PROGRAM PRG_PLAS_02_PackAggregationCtrl
VAR
	tonEnableCameraSystem					: TON;
	bEnablePackAggregationCameraSystem	: BOOL;
	bEnablePackTriggeringAfterDelay			: BOOL;

	tofPackAggregationCameraOFFDelay 		: TOF;
	rsInhibitCameraTrigger				: RS;
	rtrigNewArrived						: R_TRIG;
	bNewCodeIsProccesing				: BOOL;

	tonValidationTimout					: TON;
	bValidationTimeout					: BOOL;
	bValidationTimeoutReset				: BOOL;

	(*stPackAggregationCameraOptions		: ST_SCANNER_Options := (eScannerType := E_MV_420_FULL, nImageBuffer := 1, nExpectedResp := 1);*)
	fbPackAggregationCamera				: ARRAY [2..3] OF FB_SCANNER_CameraSelect;
	fbPackAggregationEvaluation			: ARRAY [2..3] OF FB_SCANNER_Evaluation;

	rtPackAggregationCameraDone		: ARRAY [2..3] OF R_TRIG;
	bPackAggregationCameraDone		: ARRAY [2..3] OF BOOL;

	fbAdd2PackToInfeedQ					: FB_T01_Add2PackToInfeedQ;
	(*bAddToPackQueueDone				: BOOL;*)

	fbDebugCNT							: FB_DEBUG_CounterArray;
	aCNTDebug							: ARRAY [1..10] OF UDINT;
	bResetCNT								: BOOL;

END_VAR
VAR // added by the converter: edge detectors and wires of the graphical bodies
    _w1 : BOOL;
    _w2 : UDINT;
END_VAR

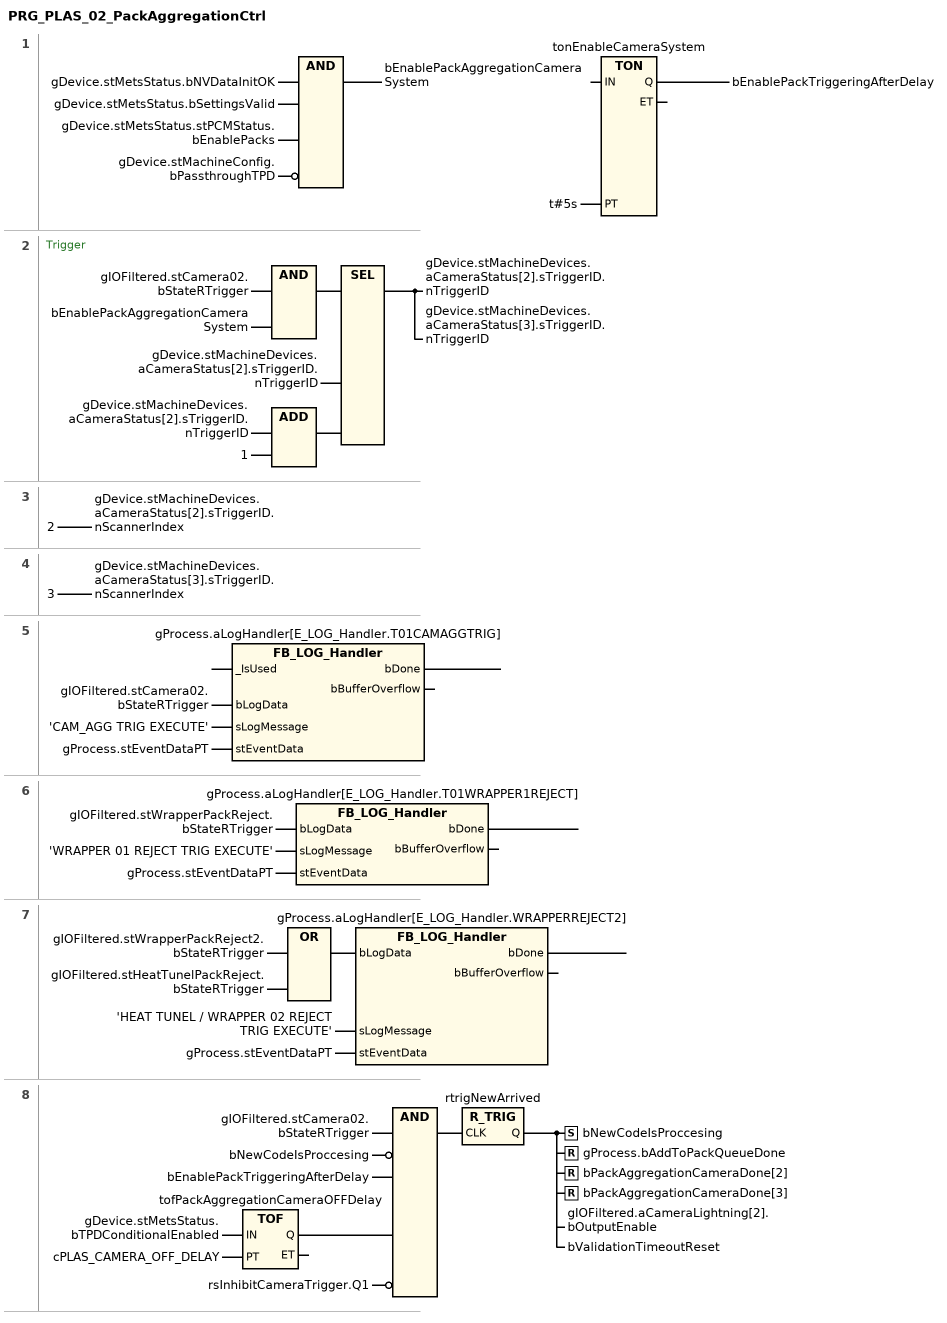
// NETWORK 1
_w1 := gDevice.stMetsStatus.bNVDataInitOK AND gDevice.stMetsStatus.bSettingsValid AND gDevice.stMetsStatus.stPCMStatus.bEnablePacks AND NOT gDevice.stMachineConfig.bPassthroughTPD;
bEnablePackAggregationCameraSystem := _w1;
tonEnableCameraSystem(IN := _w1, PT := t#5s); // TON
bEnablePackTriggeringAfterDelay := tonEnableCameraSystem.Q;

// NETWORK 2
// Trigger
_w2 := SEL(gIOFiltered.stCamera02.bStateRTrigger AND bEnablePackAggregationCameraSystem, gDevice.stMachineDevices.aCameraStatus[2].sTriggerID.nTriggerID, gDevice.stMachineDevices.aCameraStatus[2].sTriggerID.nTriggerID + 1);
gDevice.stMachineDevices.aCameraStatus[2].sTriggerID.nTriggerID := _w2;
gDevice.stMachineDevices.aCameraStatus[3].sTriggerID.nTriggerID := _w2;

// NETWORK 3
gDevice.stMachineDevices.aCameraStatus[2].sTriggerID.nScannerIndex := 2;

// NETWORK 4
gDevice.stMachineDevices.aCameraStatus[3].sTriggerID.nScannerIndex := 3;

// NETWORK 5
gProcess.aLogHandler[E_LOG_Handler.T01CAMAGGTRIG](
    bLogData := gIOFiltered.stCamera02.bStateRTrigger,
    sLogMessage := 'CAM_AGG TRIG EXECUTE',
    stEventData := gProcess.stEventDataPT); // FB_LOG_Handler

// NETWORK 6
gProcess.aLogHandler[E_LOG_Handler.T01WRAPPER1REJECT](
    bLogData := gIOFiltered.stWrapperPackReject.bStateRTrigger,
    sLogMessage := 'WRAPPER 01 REJECT TRIG EXECUTE',
    stEventData := gProcess.stEventDataPT); // FB_LOG_Handler

// NETWORK 7
gProcess.aLogHandler[E_LOG_Handler.WRAPPERREJECT2](
    bLogData := gIOFiltered.stWrapperPackReject2.bStateRTrigger OR gIOFiltered.stHeatTunelPackReject.bStateRTrigger,
    sLogMessage := 'HEAT TUNEL / WRAPPER 02 REJECT TRIG EXECUTE',
    stEventData := gProcess.stEventDataPT); // FB_LOG_Handler

// NETWORK 8
tofPackAggregationCameraOFFDelay(IN := gDevice.stMetsStatus.bTPDConditionalEnabled, PT := cPLAS_CAMERA_OFF_DELAY); // TOF
rtrigNewArrived(CLK := gIOFiltered.stCamera02.bStateRTrigger AND NOT bNewCodeIsProccesing AND bEnablePackTriggeringAfterDelay AND tofPackAggregationCameraOFFDelay.Q AND NOT rsInhibitCameraTrigger.Q1); // R_TRIG
bNewCodeIsProccesing S= rtrigNewArrived.Q;
gProcess.bAddToPackQueueDone R= rtrigNewArrived.Q;
bPackAggregationCameraDone[2] R= rtrigNewArrived.Q;
bPackAggregationCameraDone[3] R= rtrigNewArrived.Q;
gIOFiltered.aCameraLightning[2].bOutputEnable := rtrigNewArrived.Q;
bValidationTimeoutReset := rtrigNewArrived.Q;

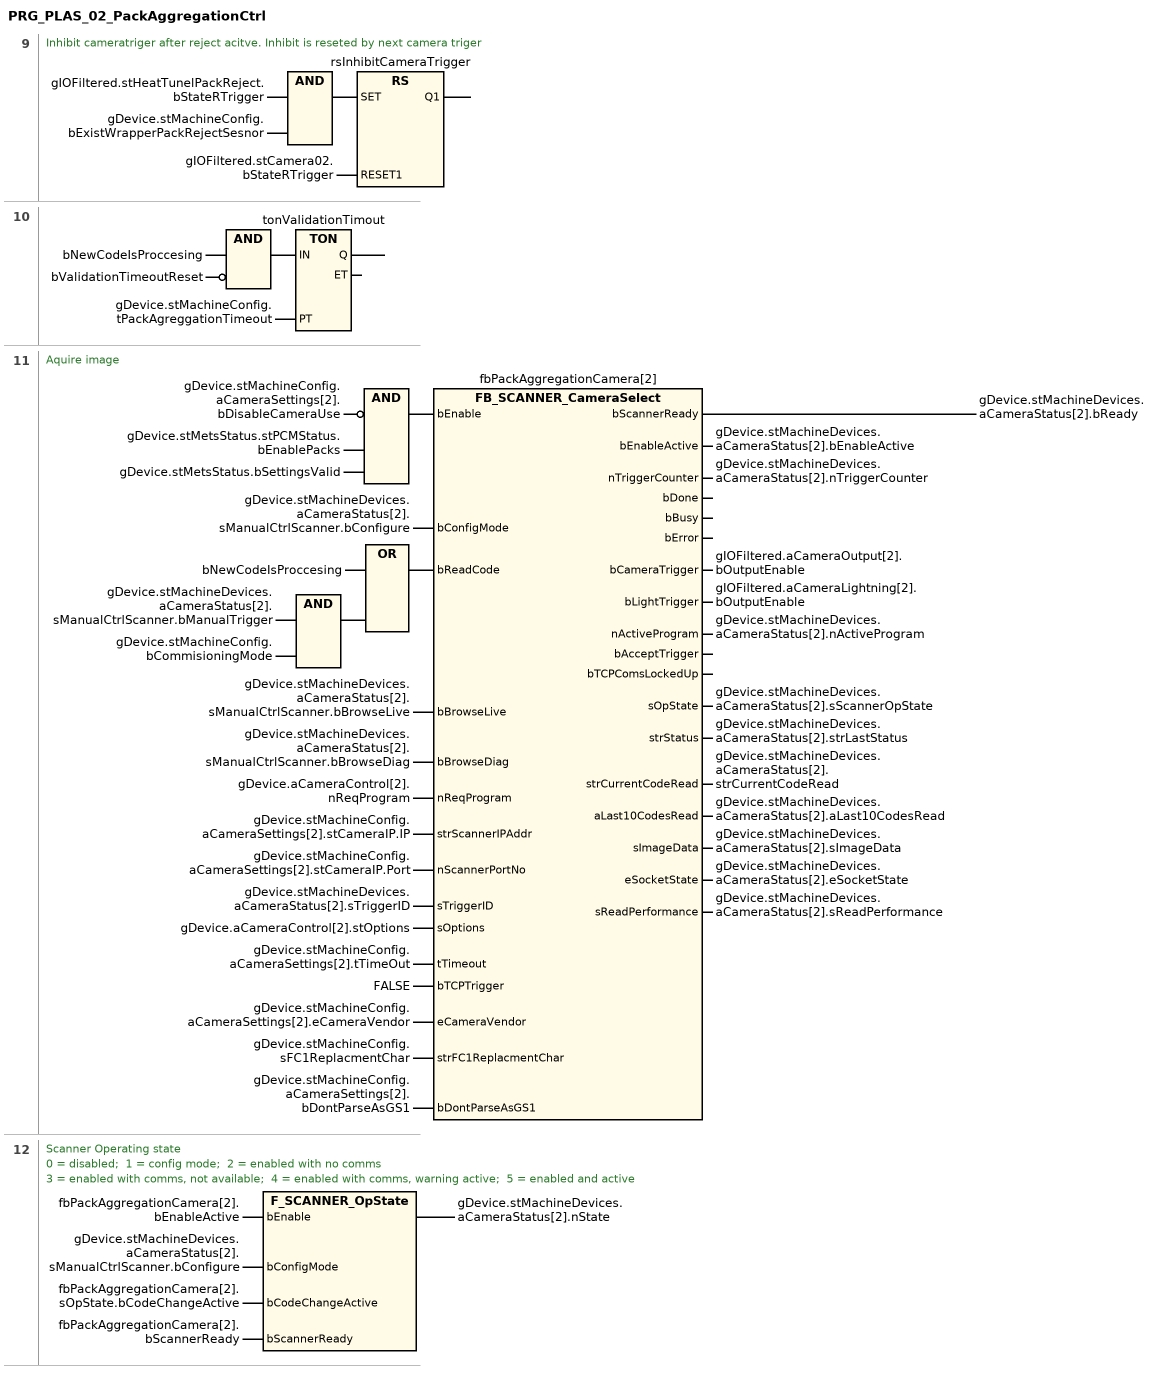
// NETWORK 9
// Inhibit cameratriger after reject acitve. Inhibit is reseted by next camera triger
rsInhibitCameraTrigger(SET := gIOFiltered.stHeatTunelPackReject.bStateRTrigger AND gDevice.stMachineConfig.bExistWrapperPackRejectSesnor, RESET1 := gIOFiltered.stCamera02.bStateRTrigger); // RS

// NETWORK 10
tonValidationTimout(IN := bNewCodeIsProccesing AND NOT bValidationTimeoutReset, PT := gDevice.stMachineConfig.tPackAgreggationTimeout); // TON

// NETWORK 11
// Aquire image
fbPackAggregationCamera[2](
    bEnable := NOT gDevice.stMachineConfig.aCameraSettings[2].bDisableCameraUse AND gDevice.stMetsStatus.stPCMStatus.bEnablePacks AND gDevice.stMetsStatus.bSettingsValid,
    bConfigMode := gDevice.stMachineDevices.aCameraStatus[2].sManualCtrlScanner.bConfigure,
    bReadCode := bNewCodeIsProccesing OR gDevice.stMachineDevices.aCameraStatus[2].sManualCtrlScanner.bManualTrigger AND gDevice.stMachineConfig.bCommisioningMode,
    bBrowseLive := gDevice.stMachineDevices.aCameraStatus[2].sManualCtrlScanner.bBrowseLive,
    bBrowseDiag := gDevice.stMachineDevices.aCameraStatus[2].sManualCtrlScanner.bBrowseDiag,
    nReqProgram := gDevice.aCameraControl[2].nReqProgram,
    strScannerIPAddr := gDevice.stMachineConfig.aCameraSettings[2].stCameraIP.IP,
    nScannerPortNo := gDevice.stMachineConfig.aCameraSettings[2].stCameraIP.Port,
    sTriggerID := gDevice.stMachineDevices.aCameraStatus[2].sTriggerID,
    sOptions := gDevice.aCameraControl[2].stOptions,
    tTimeout := gDevice.stMachineConfig.aCameraSettings[2].tTimeOut,
    bTCPTrigger := FALSE,
    eCameraVendor := gDevice.stMachineConfig.aCameraSettings[2].eCameraVendor,
    strFC1ReplacmentChar := gDevice.stMachineConfig.sFC1ReplacmentChar,
    bDontParseAsGS1 := gDevice.stMachineConfig.aCameraSettings[2].bDontParseAsGS1,
    bEnableActive => gDevice.stMachineDevices.aCameraStatus[2].bEnableActive,
    nTriggerCounter => gDevice.stMachineDevices.aCameraStatus[2].nTriggerCounter,
    bCameraTrigger => gIOFiltered.aCameraOutput[2].bOutputEnable,
    bLightTrigger => gIOFiltered.aCameraLightning[2].bOutputEnable,
    nActiveProgram => gDevice.stMachineDevices.aCameraStatus[2].nActiveProgram,
    sOpState => gDevice.stMachineDevices.aCameraStatus[2].sScannerOpState,
    strStatus => gDevice.stMachineDevices.aCameraStatus[2].strLastStatus,
    strCurrentCodeRead => gDevice.stMachineDevices.aCameraStatus[2].strCurrentCodeRead,
    aLast10CodesRead => gDevice.stMachineDevices.aCameraStatus[2].aLast10CodesRead,
    sImageData => gDevice.stMachineDevices.aCameraStatus[2].sImageData,
    eSocketState => gDevice.stMachineDevices.aCameraStatus[2].eSocketState,
    sReadPerformance => gDevice.stMachineDevices.aCameraStatus[2].sReadPerformance); // FB_SCANNER_CameraSelect
gDevice.stMachineDevices.aCameraStatus[2].bReady := fbPackAggregationCamera[2].bScannerReady;

// NETWORK 12
// 					Scanner Operating state
// 0 = disabled;  1 = config mode;  2 = enabled with no comms
// 3 = enabled with comms, not available;  4 = enabled with comms, warning active;  5 = enabled and active
//
gDevice.stMachineDevices.aCameraStatus[2].nState := F_SCANNER_OpState(bEnable := fbPackAggregationCamera[2].bEnableActive, bConfigMode := gDevice.stMachineDevices.aCameraStatus[2].sManualCtrlScanner.bConfigure, bCodeChangeActive := fbPackAggregationCamera[2].sOpState.bCodeChangeActive, bScannerReady := fbPackAggregationCamera[2].bScannerReady);

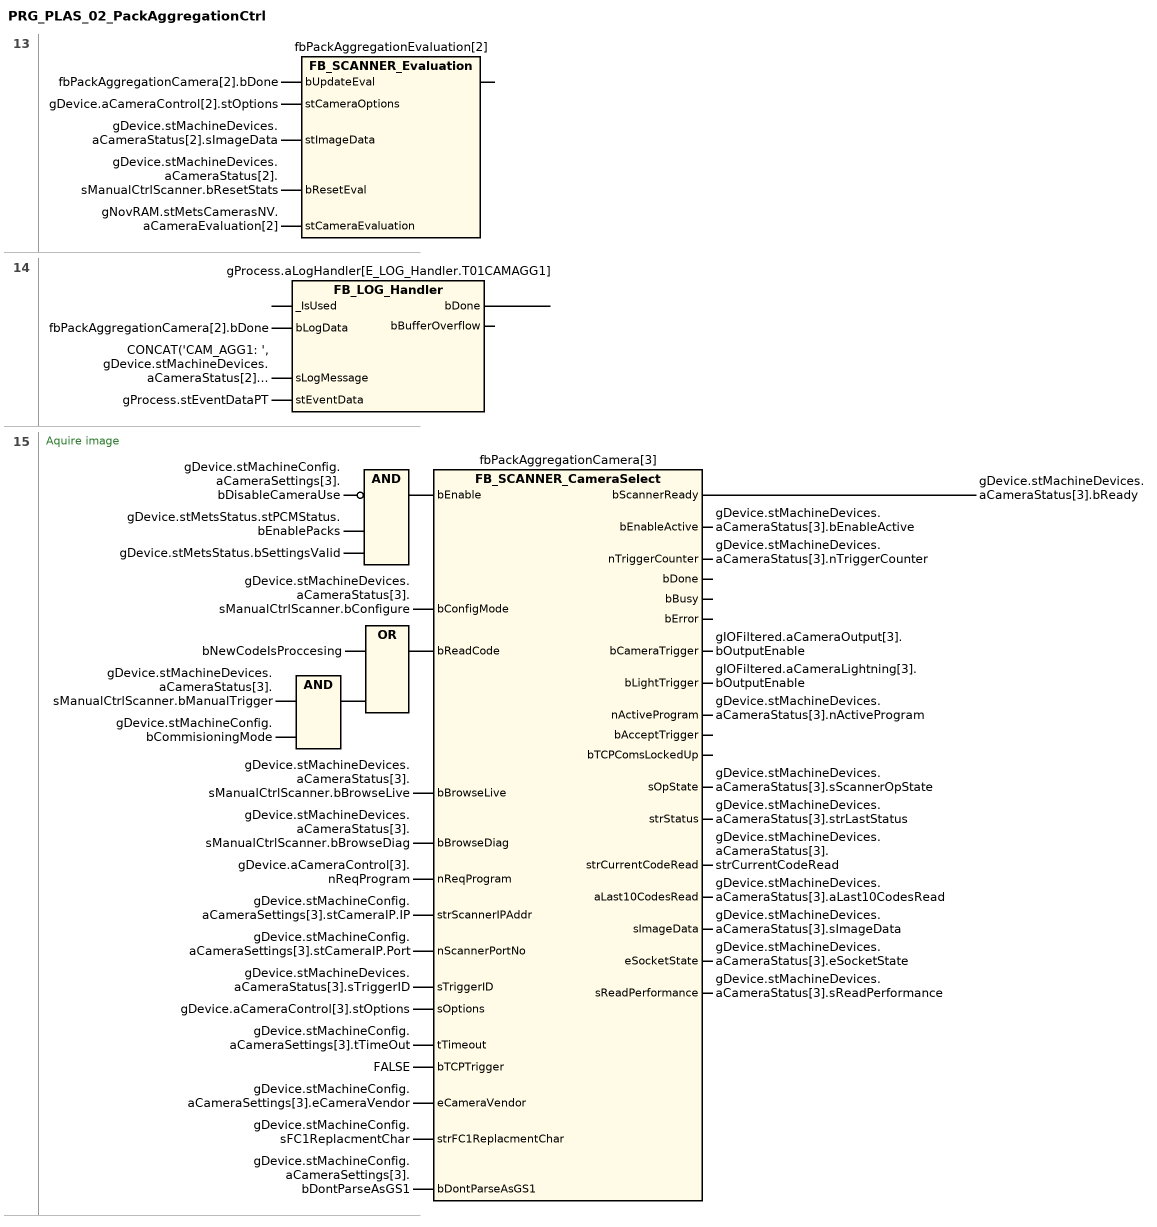
// NETWORK 13
fbPackAggregationEvaluation[2](
    bUpdateEval := fbPackAggregationCamera[2].bDone,
    stCameraOptions := gDevice.aCameraControl[2].stOptions,
    stImageData := gDevice.stMachineDevices.aCameraStatus[2].sImageData,
    bResetEval := gDevice.stMachineDevices.aCameraStatus[2].sManualCtrlScanner.bResetStats,
    stCameraEvaluation := gNovRAM.stMetsCamerasNV.aCameraEvaluation[2]); // FB_SCANNER_Evaluation

// NETWORK 14
gProcess.aLogHandler[E_LOG_Handler.T01CAMAGG1](
    bLogData := fbPackAggregationCamera[2].bDone,
    sLogMessage := CONCAT('CAM_AGG1: ', gDevice.stMachineDevices.aCameraStatus[2].strCurrentCodeRead),
    stEventData := gProcess.stEventDataPT); // FB_LOG_Handler

// NETWORK 15
// Aquire image
fbPackAggregationCamera[3](
    bEnable := NOT gDevice.stMachineConfig.aCameraSettings[3].bDisableCameraUse AND gDevice.stMetsStatus.stPCMStatus.bEnablePacks AND gDevice.stMetsStatus.bSettingsValid,
    bConfigMode := gDevice.stMachineDevices.aCameraStatus[3].sManualCtrlScanner.bConfigure,
    bReadCode := bNewCodeIsProccesing OR gDevice.stMachineDevices.aCameraStatus[3].sManualCtrlScanner.bManualTrigger AND gDevice.stMachineConfig.bCommisioningMode,
    bBrowseLive := gDevice.stMachineDevices.aCameraStatus[3].sManualCtrlScanner.bBrowseLive,
    bBrowseDiag := gDevice.stMachineDevices.aCameraStatus[3].sManualCtrlScanner.bBrowseDiag,
    nReqProgram := gDevice.aCameraControl[3].nReqProgram,
    strScannerIPAddr := gDevice.stMachineConfig.aCameraSettings[3].stCameraIP.IP,
    nScannerPortNo := gDevice.stMachineConfig.aCameraSettings[3].stCameraIP.Port,
    sTriggerID := gDevice.stMachineDevices.aCameraStatus[3].sTriggerID,
    sOptions := gDevice.aCameraControl[3].stOptions,
    tTimeout := gDevice.stMachineConfig.aCameraSettings[3].tTimeOut,
    bTCPTrigger := FALSE,
    eCameraVendor := gDevice.stMachineConfig.aCameraSettings[3].eCameraVendor,
    strFC1ReplacmentChar := gDevice.stMachineConfig.sFC1ReplacmentChar,
    bDontParseAsGS1 := gDevice.stMachineConfig.aCameraSettings[3].bDontParseAsGS1,
    bEnableActive => gDevice.stMachineDevices.aCameraStatus[3].bEnableActive,
    nTriggerCounter => gDevice.stMachineDevices.aCameraStatus[3].nTriggerCounter,
    bCameraTrigger => gIOFiltered.aCameraOutput[3].bOutputEnable,
    bLightTrigger => gIOFiltered.aCameraLightning[3].bOutputEnable,
    nActiveProgram => gDevice.stMachineDevices.aCameraStatus[3].nActiveProgram,
    sOpState => gDevice.stMachineDevices.aCameraStatus[3].sScannerOpState,
    strStatus => gDevice.stMachineDevices.aCameraStatus[3].strLastStatus,
    strCurrentCodeRead => gDevice.stMachineDevices.aCameraStatus[3].strCurrentCodeRead,
    aLast10CodesRead => gDevice.stMachineDevices.aCameraStatus[3].aLast10CodesRead,
    sImageData => gDevice.stMachineDevices.aCameraStatus[3].sImageData,
    eSocketState => gDevice.stMachineDevices.aCameraStatus[3].eSocketState,
    sReadPerformance => gDevice.stMachineDevices.aCameraStatus[3].sReadPerformance); // FB_SCANNER_CameraSelect
gDevice.stMachineDevices.aCameraStatus[3].bReady := fbPackAggregationCamera[3].bScannerReady;

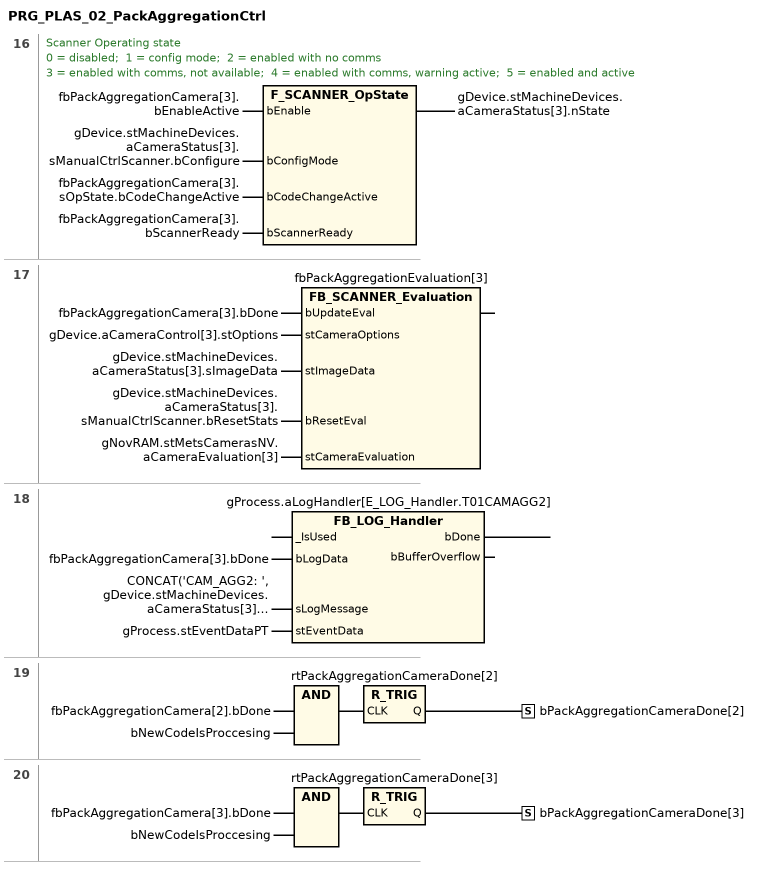
// NETWORK 16
// 					Scanner Operating state
// 0 = disabled;  1 = config mode;  2 = enabled with no comms
// 3 = enabled with comms, not available;  4 = enabled with comms, warning active;  5 = enabled and active
//
gDevice.stMachineDevices.aCameraStatus[3].nState := F_SCANNER_OpState(bEnable := fbPackAggregationCamera[3].bEnableActive, bConfigMode := gDevice.stMachineDevices.aCameraStatus[3].sManualCtrlScanner.bConfigure, bCodeChangeActive := fbPackAggregationCamera[3].sOpState.bCodeChangeActive, bScannerReady := fbPackAggregationCamera[3].bScannerReady);

// NETWORK 17
fbPackAggregationEvaluation[3](
    bUpdateEval := fbPackAggregationCamera[3].bDone,
    stCameraOptions := gDevice.aCameraControl[3].stOptions,
    stImageData := gDevice.stMachineDevices.aCameraStatus[3].sImageData,
    bResetEval := gDevice.stMachineDevices.aCameraStatus[3].sManualCtrlScanner.bResetStats,
    stCameraEvaluation := gNovRAM.stMetsCamerasNV.aCameraEvaluation[3]); // FB_SCANNER_Evaluation

// NETWORK 18
gProcess.aLogHandler[E_LOG_Handler.T01CAMAGG2](
    bLogData := fbPackAggregationCamera[3].bDone,
    sLogMessage := CONCAT('CAM_AGG2: ', gDevice.stMachineDevices.aCameraStatus[3].strCurrentCodeRead),
    stEventData := gProcess.stEventDataPT); // FB_LOG_Handler

// NETWORK 19
rtPackAggregationCameraDone[2](CLK := fbPackAggregationCamera[2].bDone AND bNewCodeIsProccesing); // R_TRIG
bPackAggregationCameraDone[2] S= rtPackAggregationCameraDone[2].Q;

// NETWORK 20
rtPackAggregationCameraDone[3](CLK := fbPackAggregationCamera[3].bDone AND bNewCodeIsProccesing); // R_TRIG
bPackAggregationCameraDone[3] S= rtPackAggregationCameraDone[3].Q;

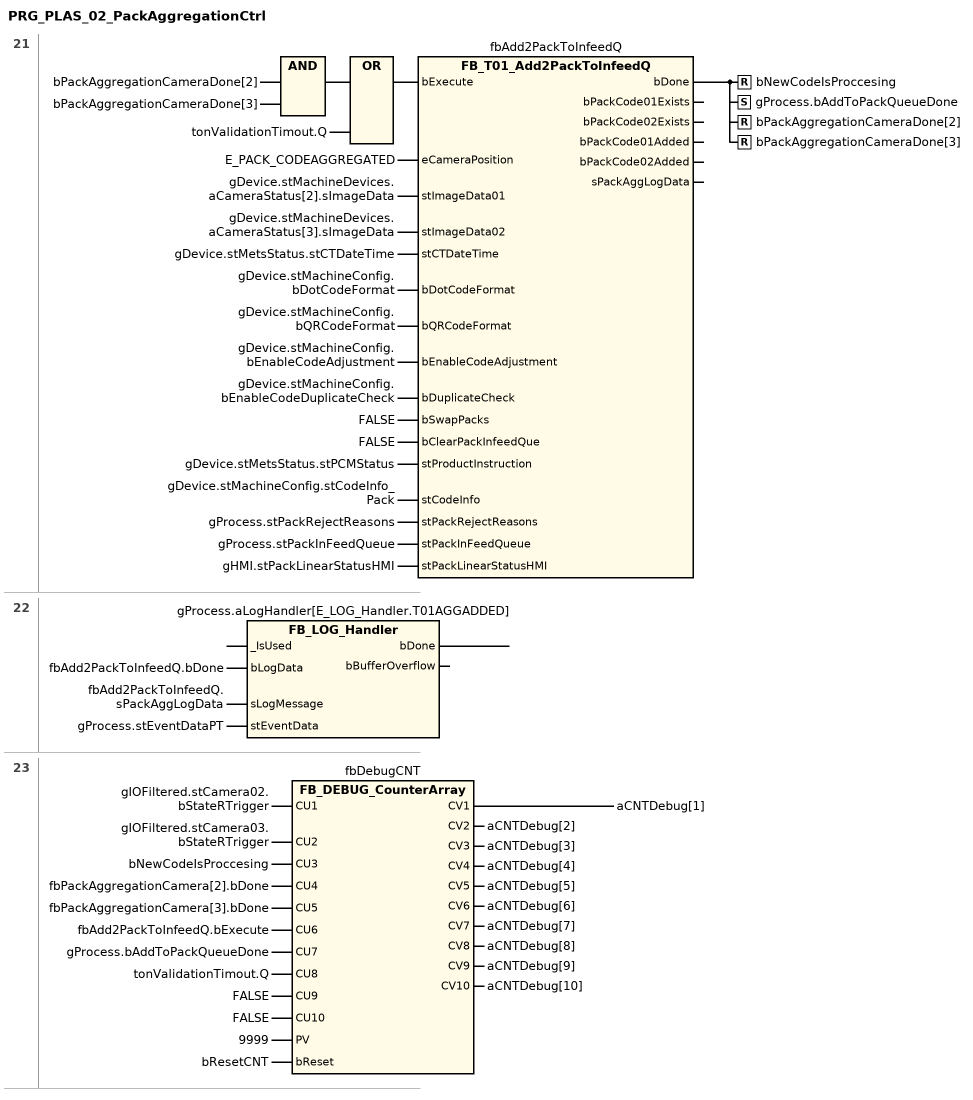
// NETWORK 21
fbAdd2PackToInfeedQ(
    bExecute := bPackAggregationCameraDone[2] AND bPackAggregationCameraDone[3] OR tonValidationTimout.Q,
    eCameraPosition := E_PACK_CODEAGGREGATED,
    stImageData01 := gDevice.stMachineDevices.aCameraStatus[2].sImageData,
    stImageData02 := gDevice.stMachineDevices.aCameraStatus[3].sImageData,
    stCTDateTime := gDevice.stMetsStatus.stCTDateTime,
    bDotCodeFormat := gDevice.stMachineConfig.bDotCodeFormat,
    bQRCodeFormat := gDevice.stMachineConfig.bQRCodeFormat,
    bEnableCodeAdjustment := gDevice.stMachineConfig.bEnableCodeAdjustment,
    bDuplicateCheck := gDevice.stMachineConfig.bEnableCodeDuplicateCheck,
    bSwapPacks := FALSE,
    bClearPackInfeedQue := FALSE,
    stProductInstruction := gDevice.stMetsStatus.stPCMStatus,
    stCodeInfo := gDevice.stMachineConfig.stCodeInfo_Pack,
    stPackRejectReasons := gProcess.stPackRejectReasons,
    stPackInFeedQueue := gProcess.stPackInFeedQueue,
    stPackLinearStatusHMI := gHMI.stPackLinearStatusHMI); // FB_T01_Add2PackToInfeedQ
bNewCodeIsProccesing R= fbAdd2PackToInfeedQ.bDone;
gProcess.bAddToPackQueueDone S= fbAdd2PackToInfeedQ.bDone;
bPackAggregationCameraDone[2] R= fbAdd2PackToInfeedQ.bDone;
bPackAggregationCameraDone[3] R= fbAdd2PackToInfeedQ.bDone;

// NETWORK 22
gProcess.aLogHandler[E_LOG_Handler.T01AGGADDED](
    bLogData := fbAdd2PackToInfeedQ.bDone,
    sLogMessage := fbAdd2PackToInfeedQ.sPackAggLogData,
    stEventData := gProcess.stEventDataPT); // FB_LOG_Handler

// NETWORK 23
fbDebugCNT(
    CU1 := gIOFiltered.stCamera02.bStateRTrigger,
    CU2 := gIOFiltered.stCamera03.bStateRTrigger,
    CU3 := bNewCodeIsProccesing,
    CU4 := fbPackAggregationCamera[2].bDone,
    CU5 := fbPackAggregationCamera[3].bDone,
    CU6 := fbAdd2PackToInfeedQ.bExecute,
    CU7 := gProcess.bAddToPackQueueDone,
    CU8 := tonValidationTimout.Q,
    CU9 := FALSE,
    CU10 := FALSE,
    PV := 9999,
    bReset := bResetCNT,
    CV2 => aCNTDebug[2],
    CV3 => aCNTDebug[3],
    CV4 => aCNTDebug[4],
    CV5 => aCNTDebug[5],
    CV6 => aCNTDebug[6],
    CV7 => aCNTDebug[7],
    CV8 => aCNTDebug[8],
    CV9 => aCNTDebug[9],
    CV10 => aCNTDebug[10]); // FB_DEBUG_CounterArray
aCNTDebug[1] := fbDebugCNT.CV1;

END_PROGRAM

(* stored: Version 1.1.0.1
   POU PRG_PLAS_02_PackAggregationCtrl: Id {db1ee7c0-94f7-40ee-a189-7e62e05cda71}, SpecialFunc None *)
